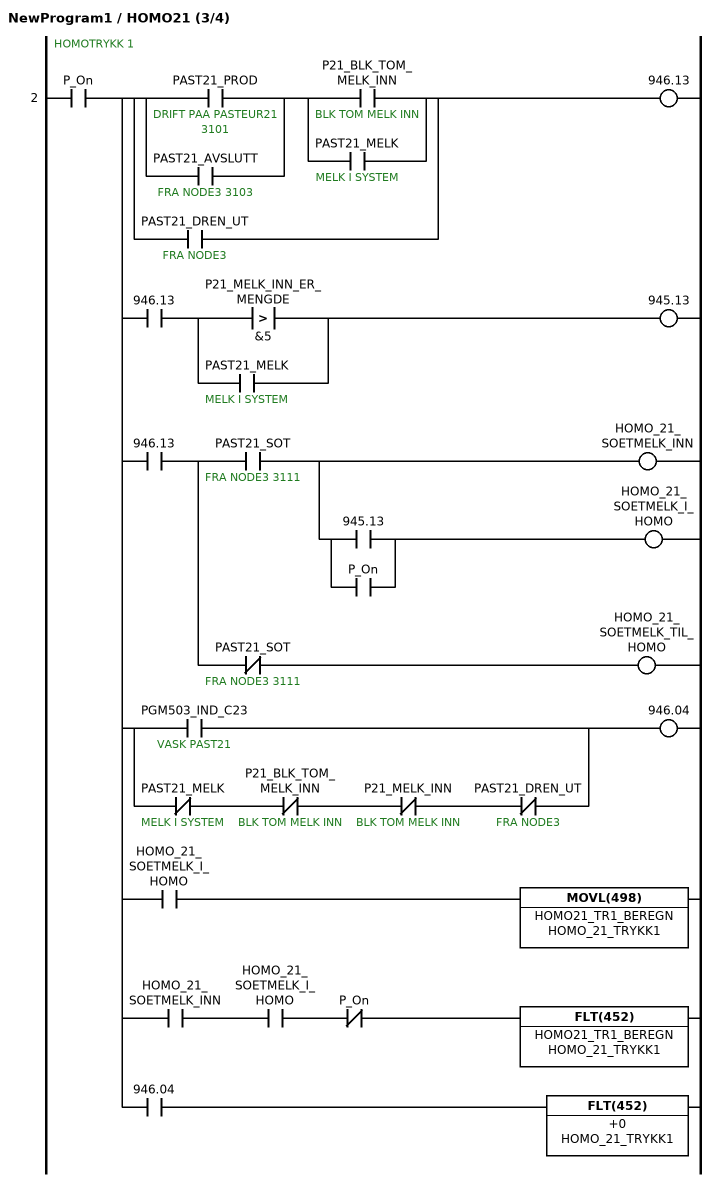
; [picture p1128: NewProgram1 / HOMO21, rungs 2-2]
; rung 2: HOMOTRYKK 1
LD P_On
OUT TR0
LD PAST21_PROD  ; DRIFT PAA PASTEUR21 3101
OR PAST21_AVSLUTT  ; FRA NODE3 3103
LD P21_BLK_TOM_MELK_INN  ; BLK TOM MELK INN
OR PAST21_MELK  ; MELK I SYSTEM
ANDLD
OR PAST21_DREN_UT  ; FRA NODE3
ANDLD
OUT 946.13
LD TR0
AND 946.13
LD>(320) P21_MELK_INN_ER_MENGDE &5
OR PAST21_MELK  ; MELK I SYSTEM
ANDLD
OUT 945.13
LD TR0
AND 946.13
OUT TR1
AND PAST21_SOT  ; FRA NODE3 3111
OUT HOMO_21_SOETMELK_INN
LD 945.13
OR P_On
ANDLD
OUT HOMO_21_SOETMELK_I_HOMO
LD TR1
ANDNOT PAST21_SOT  ; FRA NODE3 3111
OUT HOMO_21_SOETMELK_TIL_HOMO
LD TR0
LD PGM503_IND_C23  ; VASK PAST21
LDNOT PAST21_MELK  ; MELK I SYSTEM
ANDNOT P21_BLK_TOM_MELK_INN  ; BLK TOM MELK INN
ANDNOT P21_MELK_INN  ; BLK TOM MELK INN
ANDNOT PAST21_DREN_UT  ; FRA NODE3
ORLD
ANDLD
OUT 946.04
LD TR0
AND HOMO_21_SOETMELK_I_HOMO
MOVL(498) HOMO21_TR1_BEREGN HOMO_21_TRYKK1
LD TR0
AND HOMO_21_SOETMELK_INN
AND HOMO_21_SOETMELK_I_HOMO
ANDNOT P_On
FLT(452) HOMO21_TR1_BEREGN HOMO_21_TRYKK1
LD TR0
AND 946.04
FLT(452) +0 HOMO_21_TRYKK1

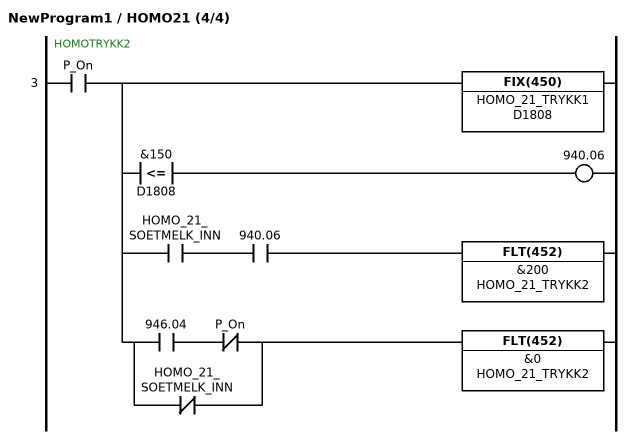
; rung 3: HOMOTRYKK2
LD P_On
OUT TR0
FIX(450) HOMO_21_TRYKK1 D1808
AND<=(315) &150 D1808
OUT 940.06
LD TR0
AND HOMO_21_SOETMELK_INN
AND 940.06
FLT(452) &200 HOMO_21_TRYKK2
LD TR0
LD 946.04
ANDNOT P_On
ORNOT HOMO_21_SOETMELK_INN
ANDLD
FLT(452) &0 HOMO_21_TRYKK2

### Section PAST22_TEMP_NIVÅ

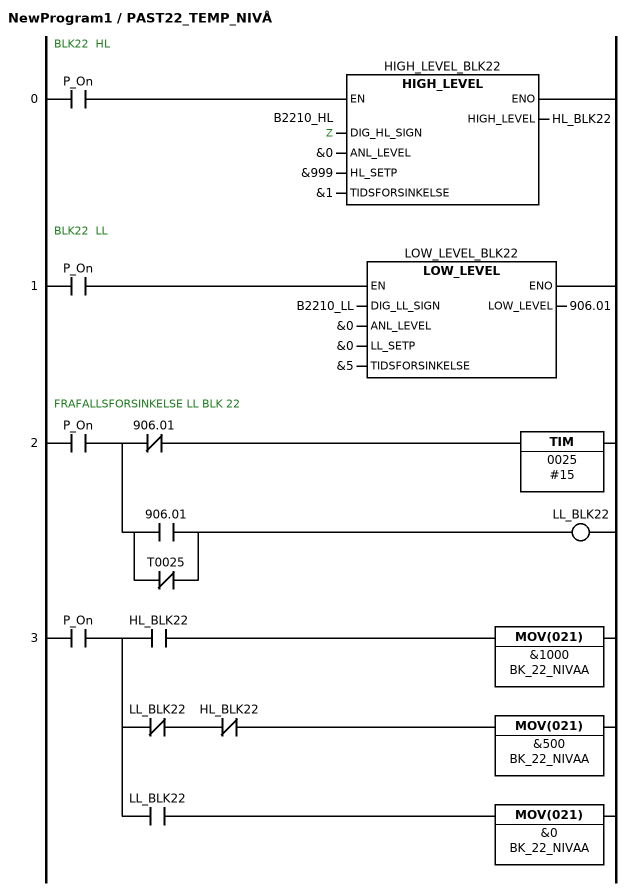
; rung 0: BLK22  HL
LD P_On
CALL HIGH_LEVEL_BLK22 : HIGH_LEVEL (DIG_HL_SIGN := B2210_HL, ANL_LEVEL := &0, HL_SETP := &999, TIDSFORSINKELSE := &1, HIGH_LEVEL => HL_BLK22)  ; Z
; rung 1: BLK22  LL
LD P_On
CALL LOW_LEVEL_BLK22 : LOW_LEVEL (DIG_LL_SIGN := B2210_LL, ANL_LEVEL := &0, LL_SETP := &0, TIDSFORSINKELSE := &5, LOW_LEVEL => 906.01)
; rung 2: FRAFALLSFORSINKELSE LL BLK 22
LD P_On
OUT TR0
ANDNOT 906.01
TIM 0025 #15
LD TR0
LD 906.01
ORNOT T0025
ANDLD
OUT LL_BLK22
; rung 3
LD P_On
OUT TR0
AND HL_BLK22
MOV(021) &1000 BK_22_NIVAA
LD TR0
ANDNOT LL_BLK22
ANDNOT HL_BLK22
MOV(021) &500 BK_22_NIVAA
LD TR0
AND LL_BLK22
MOV(021) &0 BK_22_NIVAA

### Section PAST22_DRIFT_OG_TYPE_MELK

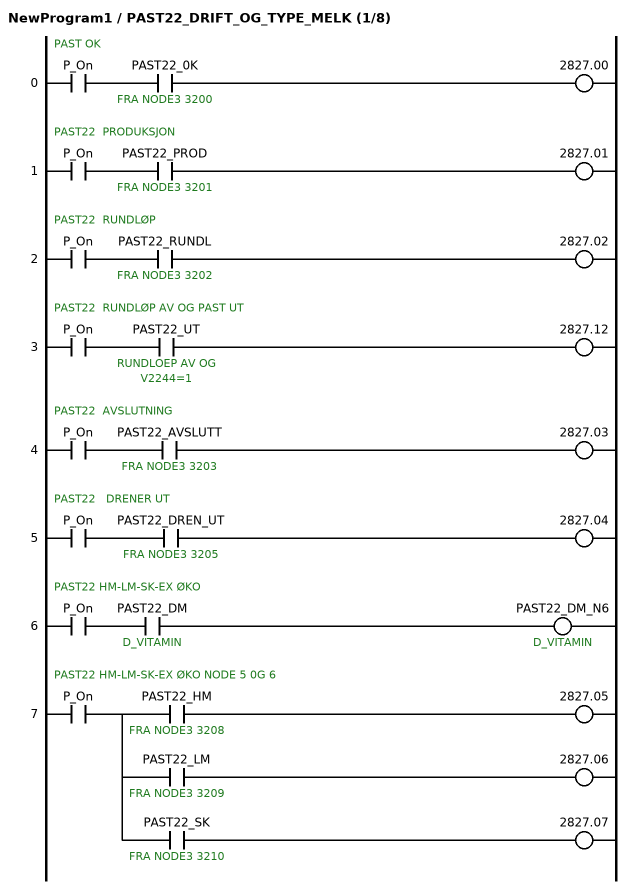
; rung 0: PAST OK
LD P_On
AND PAST22_0K  ; FRA NODE3 3200
OUT 2827.00
; rung 1: PAST22  PRODUKSJON
LD P_On
AND PAST22_PROD  ; FRA NODE3 3201
OUT 2827.01
; rung 2: PAST22  RUNDLØP
LD P_On
AND PAST22_RUNDL  ; FRA NODE3 3202
OUT 2827.02
; rung 3: PAST22  RUNDLØP AV OG PAST UT
LD P_On
AND PAST22_UT  ; RUNDLOEP AV OG V2244=1
OUT 2827.12
; rung 4: PAST22  AVSLUTNING
LD P_On
AND PAST22_AVSLUTT  ; FRA NODE3 3203
OUT 2827.03
; rung 5: PAST22   DRENER UT
LD P_On
AND PAST22_DREN_UT  ; FRA NODE3 3205
OUT 2827.04
; rung 6: PAST22 HM-LM-SK-EX ØKO
LD P_On
AND PAST22_DM  ; D_VITAMIN
OUT PAST22_DM_N6  ; D_VITAMIN
; rung 7: PAST22 HM-LM-SK-EX ØKO NODE 5 0G 6
LD P_On
OUT TR0
AND PAST22_HM  ; FRA NODE3 3208
OUT 2827.05
LD TR0
AND PAST22_LM  ; FRA NODE3 3209
OUT 2827.06
LD TR0
AND PAST22_SK  ; FRA NODE3 3210
OUT 2827.07

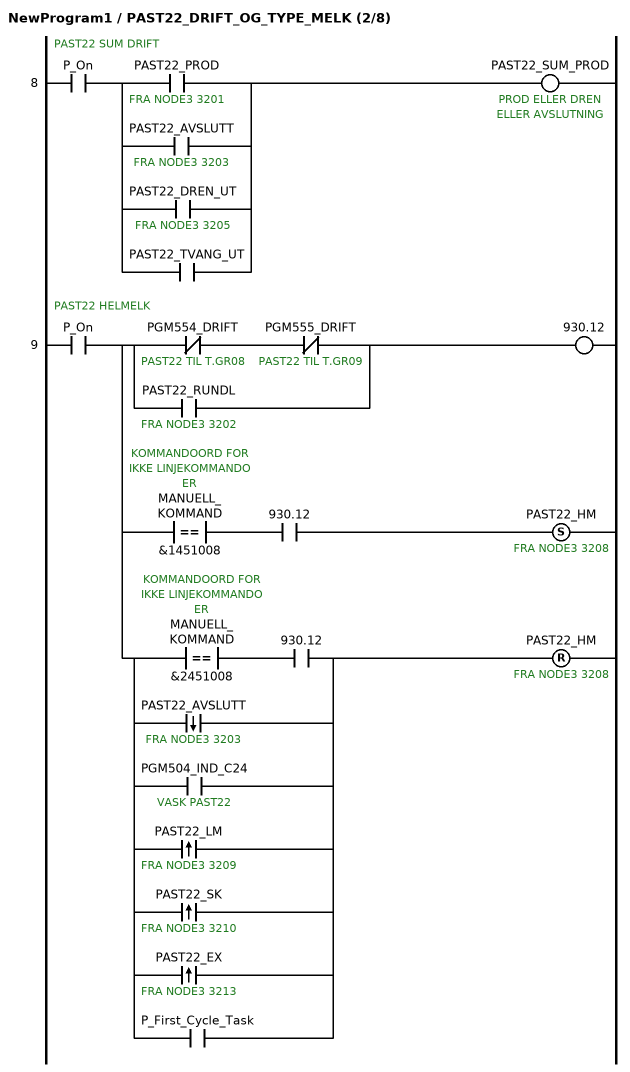
; rung 8: PAST22 SUM DRIFT
LD P_On
LD PAST22_PROD  ; FRA NODE3 3201
OR PAST22_AVSLUTT  ; FRA NODE3 3203
OR PAST22_DREN_UT  ; FRA NODE3 3205
OR PAST22_TVANG_UT
ANDLD
OUT PAST22_SUM_PROD  ; PROD ELLER DREN ELLER AVSLUTNING
; rung 9: PAST22 HELMELK
LD P_On
OUT TR0
LDNOT PGM554_DRIFT  ; PAST22 TIL T.GR08
ANDNOT PGM555_DRIFT  ; PAST22 TIL T.GR09
OR PAST22_RUNDL  ; FRA NODE3 3202
ANDLD
OUT 930.12
LD TR0
AND=L(301) MANUELL_KOMMAND &1451008  ; KOMMANDOORD FOR IKKE LINJEKOMMANDOER
AND 930.12
SET PAST22_HM  ; FRA NODE3 3208
LD TR0
LD=L(301) MANUELL_KOMMAND &2451008  ; KOMMANDOORD FOR IKKE LINJEKOMMANDOER
AND 930.12
%OR PAST22_AVSLUTT  ; FRA NODE3 3203
OR PGM504_IND_C24  ; VASK PAST22
@OR PAST22_LM  ; FRA NODE3 3209
@OR PAST22_SK  ; FRA NODE3 3210
@OR PAST22_EX  ; FRA NODE3 3213
OR P_First_Cycle_Task
ANDLD
RSET PAST22_HM  ; FRA NODE3 3208

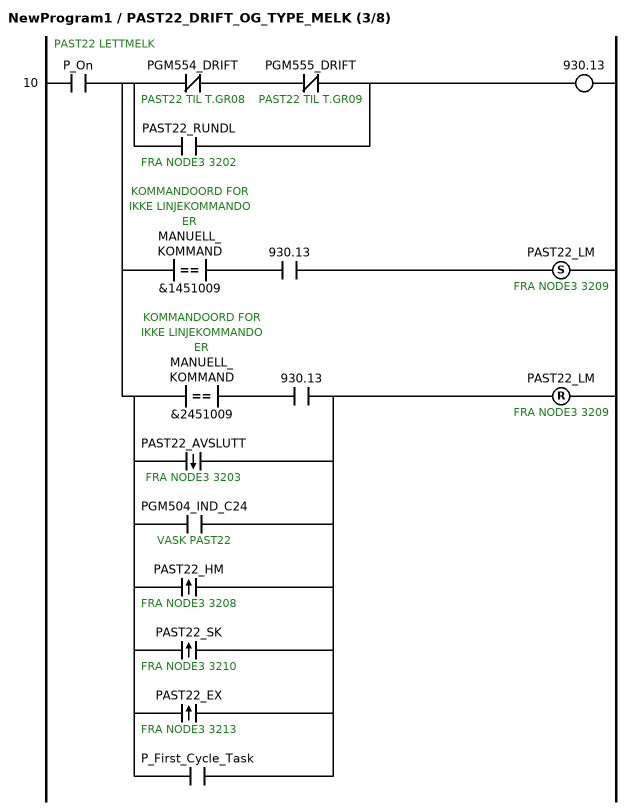
; rung 10: PAST22 LETTMELK
LD P_On
OUT TR0
LDNOT PGM554_DRIFT  ; PAST22 TIL T.GR08
ANDNOT PGM555_DRIFT  ; PAST22 TIL T.GR09
OR PAST22_RUNDL  ; FRA NODE3 3202
ANDLD
OUT 930.13
LD TR0
AND=L(301) MANUELL_KOMMAND &1451009  ; KOMMANDOORD FOR IKKE LINJEKOMMANDOER
AND 930.13
SET PAST22_LM  ; FRA NODE3 3209
LD TR0
LD=L(301) MANUELL_KOMMAND &2451009  ; KOMMANDOORD FOR IKKE LINJEKOMMANDOER
AND 930.13
%OR PAST22_AVSLUTT  ; FRA NODE3 3203
OR PGM504_IND_C24  ; VASK PAST22
@OR PAST22_HM  ; FRA NODE3 3208
@OR PAST22_SK  ; FRA NODE3 3210
@OR PAST22_EX  ; FRA NODE3 3213
OR P_First_Cycle_Task
ANDLD
RSET PAST22_LM  ; FRA NODE3 3209

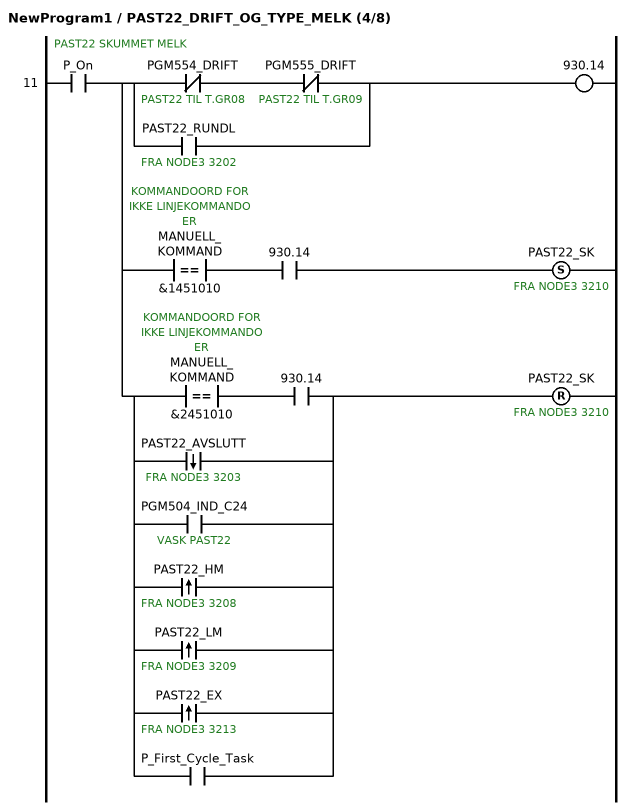
; rung 11: PAST22 SKUMMET MELK
LD P_On
OUT TR0
LDNOT PGM554_DRIFT  ; PAST22 TIL T.GR08
ANDNOT PGM555_DRIFT  ; PAST22 TIL T.GR09
OR PAST22_RUNDL  ; FRA NODE3 3202
ANDLD
OUT 930.14
LD TR0
AND=L(301) MANUELL_KOMMAND &1451010  ; KOMMANDOORD FOR IKKE LINJEKOMMANDOER
AND 930.14
SET PAST22_SK  ; FRA NODE3 3210
LD TR0
LD=L(301) MANUELL_KOMMAND &2451010  ; KOMMANDOORD FOR IKKE LINJEKOMMANDOER
AND 930.14
%OR PAST22_AVSLUTT  ; FRA NODE3 3203
OR PGM504_IND_C24  ; VASK PAST22
@OR PAST22_HM  ; FRA NODE3 3208
@OR PAST22_LM  ; FRA NODE3 3209
@OR PAST22_EX  ; FRA NODE3 3213
OR P_First_Cycle_Task
ANDLD
RSET PAST22_SK  ; FRA NODE3 3210

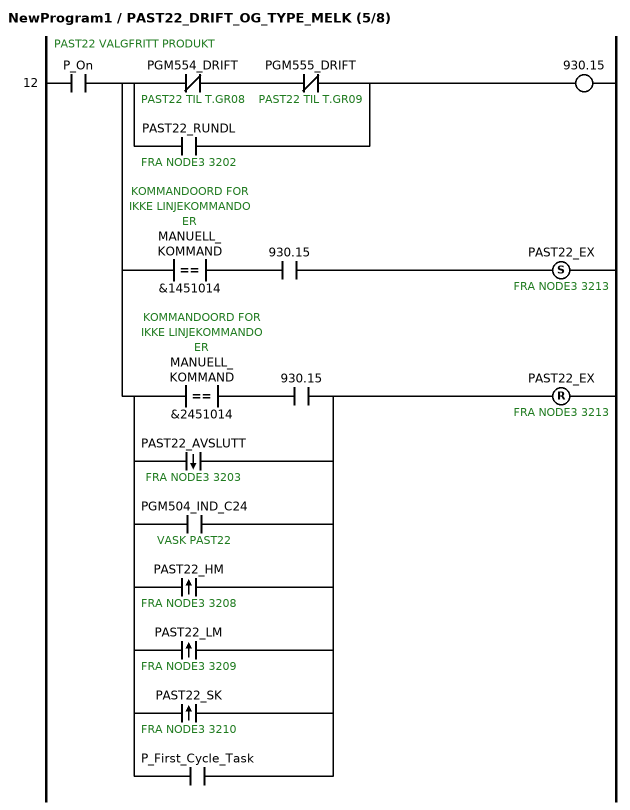
; rung 12: PAST22 VALGFRITT PRODUKT
LD P_On
OUT TR0
LDNOT PGM554_DRIFT  ; PAST22 TIL T.GR08
ANDNOT PGM555_DRIFT  ; PAST22 TIL T.GR09
OR PAST22_RUNDL  ; FRA NODE3 3202
ANDLD
OUT 930.15
LD TR0
AND=L(301) MANUELL_KOMMAND &1451014  ; KOMMANDOORD FOR IKKE LINJEKOMMANDOER
AND 930.15
SET PAST22_EX  ; FRA NODE3 3213
LD TR0
LD=L(301) MANUELL_KOMMAND &2451014  ; KOMMANDOORD FOR IKKE LINJEKOMMANDOER
AND 930.15
%OR PAST22_AVSLUTT  ; FRA NODE3 3203
OR PGM504_IND_C24  ; VASK PAST22
@OR PAST22_HM  ; FRA NODE3 3208
@OR PAST22_LM  ; FRA NODE3 3209
@OR PAST22_SK  ; FRA NODE3 3210
OR P_First_Cycle_Task
ANDLD
RSET PAST22_EX  ; FRA NODE3 3213

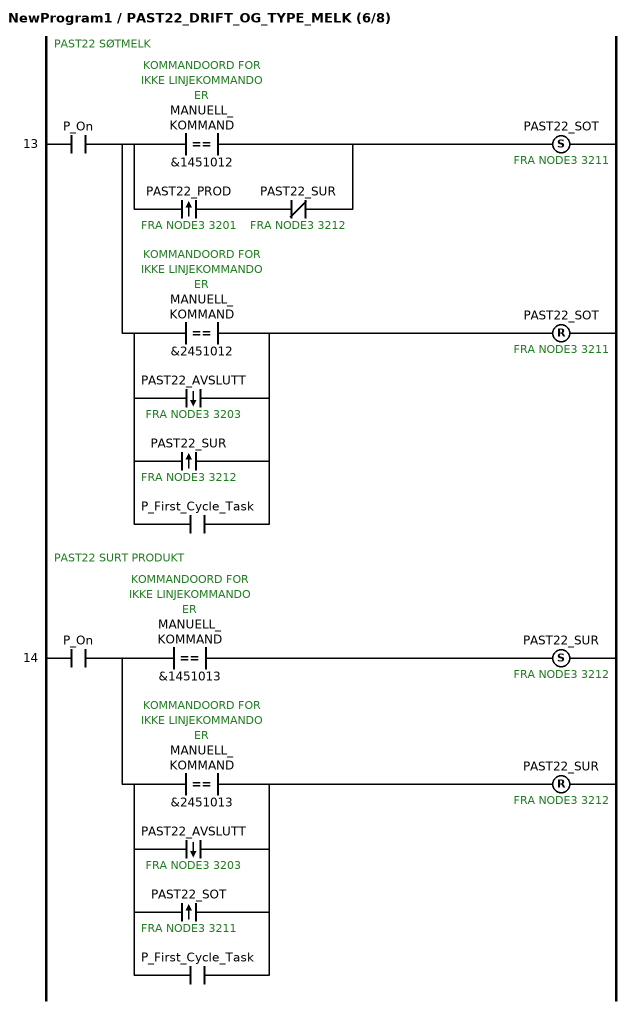
; rung 13: PAST22 SØTMELK
LD P_On
OUT TR0
LD=L(301) MANUELL_KOMMAND &1451012  ; KOMMANDOORD FOR IKKE LINJEKOMMANDOER
@LD PAST22_PROD  ; FRA NODE3 3201
ANDNOT PAST22_SUR  ; FRA NODE3 3212
ORLD
ANDLD
SET PAST22_SOT  ; FRA NODE3 3211
LD TR0
LD=L(301) MANUELL_KOMMAND &2451012  ; KOMMANDOORD FOR IKKE LINJEKOMMANDOER
%OR PAST22_AVSLUTT  ; FRA NODE3 3203
@OR PAST22_SUR  ; FRA NODE3 3212
OR P_First_Cycle_Task
ANDLD
RSET PAST22_SOT  ; FRA NODE3 3211
; rung 14: PAST22 SURT PRODUKT
LD P_On
OUT TR0
AND=L(301) MANUELL_KOMMAND &1451013  ; KOMMANDOORD FOR IKKE LINJEKOMMANDOER
SET PAST22_SUR  ; FRA NODE3 3212
LD TR0
LD=L(301) MANUELL_KOMMAND &2451013  ; KOMMANDOORD FOR IKKE LINJEKOMMANDOER
%OR PAST22_AVSLUTT  ; FRA NODE3 3203
@OR PAST22_SOT  ; FRA NODE3 3211
OR P_First_Cycle_Task
ANDLD
RSET PAST22_SUR  ; FRA NODE3 3212

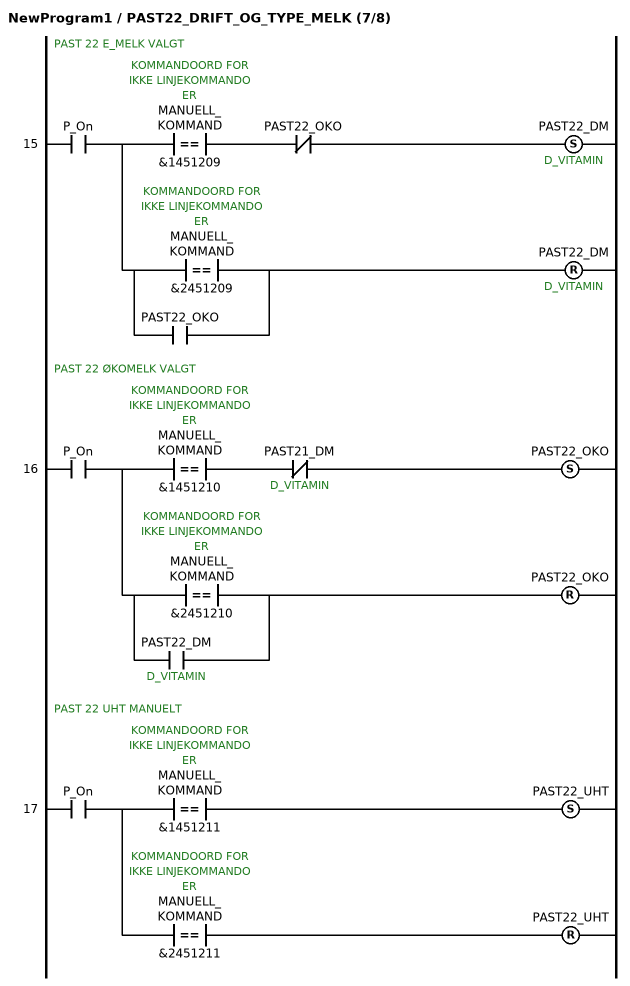
; rung 15: PAST 22 E_MELK VALGT
LD P_On
OUT TR0
AND=L(301) MANUELL_KOMMAND &1451209  ; KOMMANDOORD FOR IKKE LINJEKOMMANDOER
ANDNOT PAST22_OKO
SET PAST22_DM  ; D_VITAMIN
LD TR0
LD=L(301) MANUELL_KOMMAND &2451209  ; KOMMANDOORD FOR IKKE LINJEKOMMANDOER
OR PAST22_OKO
ANDLD
RSET PAST22_DM  ; D_VITAMIN
; rung 16: PAST 22 ØKOMELK VALGT
LD P_On
OUT TR0
AND=L(301) MANUELL_KOMMAND &1451210  ; KOMMANDOORD FOR IKKE LINJEKOMMANDOER
ANDNOT PAST21_DM  ; D_VITAMIN
SET PAST22_OKO
LD TR0
LD=L(301) MANUELL_KOMMAND &2451210  ; KOMMANDOORD FOR IKKE LINJEKOMMANDOER
OR PAST22_DM  ; D_VITAMIN
ANDLD
RSET PAST22_OKO
; rung 17: PAST 22 UHT MANUELT
LD P_On
OUT TR0
AND=L(301) MANUELL_KOMMAND &1451211  ; KOMMANDOORD FOR IKKE LINJEKOMMANDOER
SET PAST22_UHT
LD TR0
AND=L(301) MANUELL_KOMMAND &2451211  ; KOMMANDOORD FOR IKKE LINJEKOMMANDOER
RSET PAST22_UHT

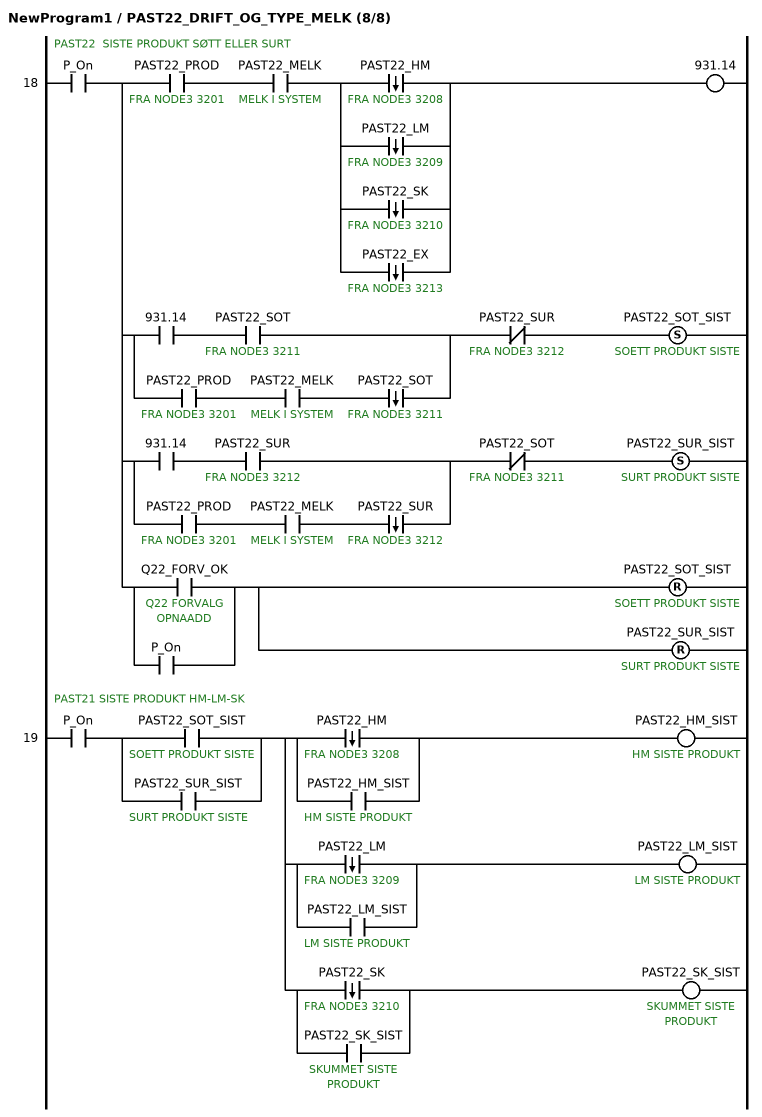
; rung 18: PAST22  SISTE PRODUKT SØTT ELLER SURT
LD P_On
OUT TR0
AND PAST22_PROD  ; FRA NODE3 3201
AND PAST22_MELK  ; MELK I SYSTEM
%LD PAST22_HM  ; FRA NODE3 3208
%OR PAST22_LM  ; FRA NODE3 3209
%OR PAST22_SK  ; FRA NODE3 3210
%OR PAST22_EX  ; FRA NODE3 3213
ANDLD
OUT 931.14
LD TR0
LD 931.14
AND PAST22_SOT  ; FRA NODE3 3211
LD PAST22_PROD  ; FRA NODE3 3201
AND PAST22_MELK  ; MELK I SYSTEM
%AND PAST22_SOT  ; FRA NODE3 3211
ORLD
ANDLD
ANDNOT PAST22_SUR  ; FRA NODE3 3212
SET PAST22_SOT_SIST  ; SOETT PRODUKT SISTE
LD TR0
LD 931.14
AND PAST22_SUR  ; FRA NODE3 3212
LD PAST22_PROD  ; FRA NODE3 3201
AND PAST22_MELK  ; MELK I SYSTEM
%AND PAST22_SUR  ; FRA NODE3 3212
ORLD
ANDLD
ANDNOT PAST22_SOT  ; FRA NODE3 3211
SET PAST22_SUR_SIST  ; SURT PRODUKT SISTE
LD TR0
LD Q22_FORV_OK  ; Q22 FORVALG OPNAADD
OR P_On
ANDLD
RSET PAST22_SOT_SIST  ; SOETT PRODUKT SISTE
RSET PAST22_SUR_SIST  ; SURT PRODUKT SISTE
; rung 19: PAST21 SISTE PRODUKT HM-LM-SK
LD P_On
LD PAST22_SOT_SIST  ; SOETT PRODUKT SISTE
OR PAST22_SUR_SIST  ; SURT PRODUKT SISTE
ANDLD
OUT TR0
%LD PAST22_HM  ; FRA NODE3 3208
OR PAST22_HM_SIST  ; HM SISTE PRODUKT
ANDLD
OUT PAST22_HM_SIST  ; HM SISTE PRODUKT
LD TR0
%LD PAST22_LM  ; FRA NODE3 3209
OR PAST22_LM_SIST  ; LM SISTE PRODUKT
ANDLD
OUT PAST22_LM_SIST  ; LM SISTE PRODUKT
LD TR0
%LD PAST22_SK  ; FRA NODE3 3210
OR PAST22_SK_SIST  ; SKUMMET SISTE PRODUKT
ANDLD
OUT PAST22_SK_SIST  ; SKUMMET SISTE PRODUKT

### Section PAST22_STATUSKONTROLL

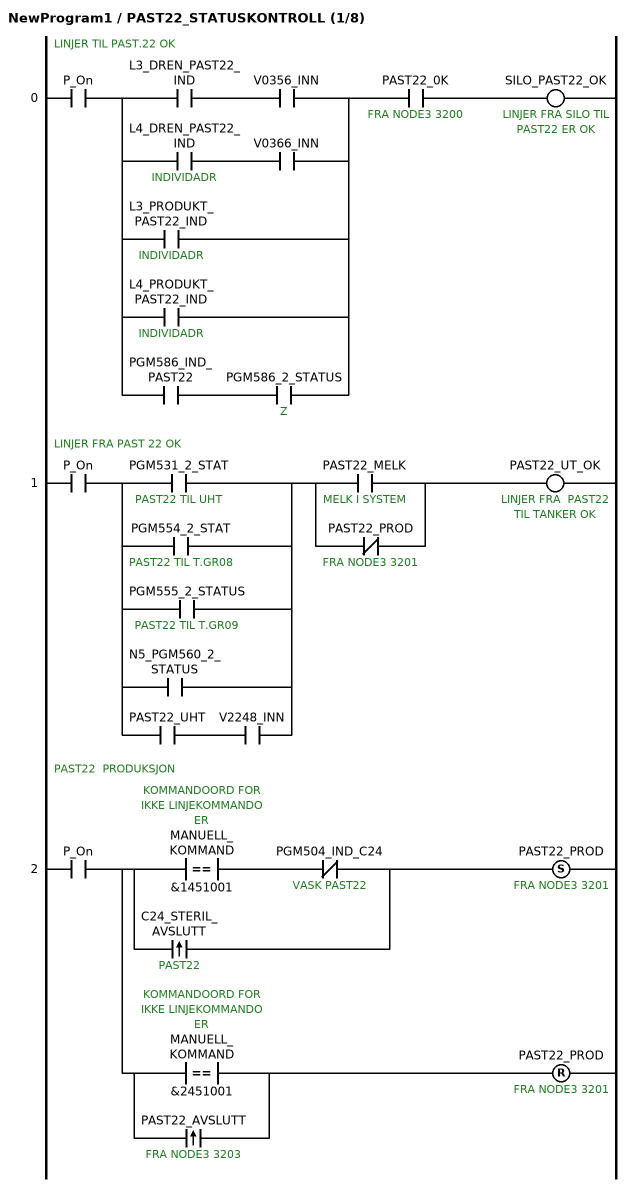
; rung 0: LINJER TIL PAST.22 OK
LD P_On
LD L3_DREN_PAST22_IND
AND V0356_INN
LD L4_DREN_PAST22_IND  ; INDIVIDADR
AND V0366_INN
ORLD
OR L3_PRODUKT_PAST22_IND  ; INDIVIDADR
OR L4_PRODUKT_PAST22_IND  ; INDIVIDADR
LD PGM586_IND_PAST22
AND PGM586_2_STATUS  ; Z
ORLD
ANDLD
AND PAST22_0K  ; FRA NODE3 3200
OUT SILO_PAST22_OK  ; LINJER FRA SILO TIL  PAST22 ER OK
; rung 1: LINJER FRA PAST 22 OK
LD P_On
LD PGM531_2_STAT  ; PAST22 TIL UHT
OR PGM554_2_STAT  ; PAST22 TIL T.GR08
OR PGM555_2_STATUS  ; PAST22 TIL T.GR09
OR N5_PGM560_2_STATUS
LD PAST22_UHT
AND V2248_INN
ORLD
ANDLD
LD PAST22_MELK  ; MELK I SYSTEM
ORNOT PAST22_PROD  ; FRA NODE3 3201
ANDLD
OUT PAST22_UT_OK  ; LINJER FRA  PAST22 TIL TANKER OK
; rung 2: PAST22  PRODUKSJON
LD P_On
OUT TR0
LD=L(301) MANUELL_KOMMAND &1451001  ; KOMMANDOORD FOR IKKE LINJEKOMMANDOER
ANDNOT PGM504_IND_C24  ; VASK PAST22
@OR C24_STERIL_AVSLUTT  ; PAST22
ANDLD
SET PAST22_PROD  ; FRA NODE3 3201
LD TR0
LD=L(301) MANUELL_KOMMAND &2451001  ; KOMMANDOORD FOR IKKE LINJEKOMMANDOER
@OR PAST22_AVSLUTT  ; FRA NODE3 3203
ANDLD
RSET PAST22_PROD  ; FRA NODE3 3201

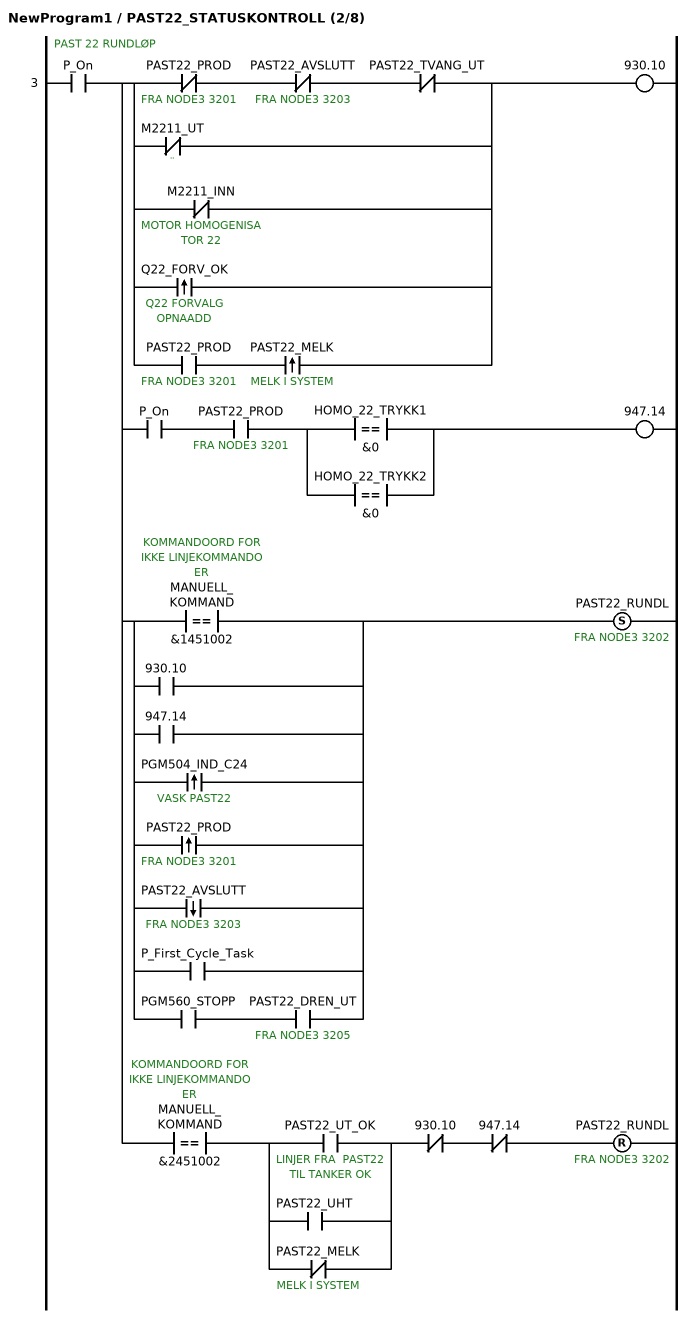
; rung 3: PAST 22 RUNDLØP
LD P_On
OUT TR0
LDNOT PAST22_PROD  ; FRA NODE3 3201
ANDNOT PAST22_AVSLUTT  ; FRA NODE3 3203
ANDNOT PAST22_TVANG_UT
ORNOT M2211_UT  ; ¨
ORNOT M2211_INN  ; MOTOR HOMOGENISATOR 22
@OR Q22_FORV_OK  ; Q22 FORVALG OPNAADD
LD PAST22_PROD  ; FRA NODE3 3201
@AND PAST22_MELK  ; MELK I SYSTEM
ORLD
ANDLD
OUT 930.10
LD TR0
AND P_On
AND PAST22_PROD  ; FRA NODE3 3201
LD=L(301) HOMO_22_TRYKK1 &0
OR=L(301) HOMO_22_TRYKK2 &0
ANDLD
OUT 947.14
LD TR0
LD=L(301) MANUELL_KOMMAND &1451002  ; KOMMANDOORD FOR IKKE LINJEKOMMANDOER
OR 930.10
OR 947.14
@OR PGM504_IND_C24  ; VASK PAST22
@OR PAST22_PROD  ; FRA NODE3 3201
%OR PAST22_AVSLUTT  ; FRA NODE3 3203
OR P_First_Cycle_Task
LD PGM560_STOPP
AND PAST22_DREN_UT  ; FRA NODE3 3205
ORLD
ANDLD
SET PAST22_RUNDL  ; FRA NODE3 3202
LD TR0
AND=L(301) MANUELL_KOMMAND &2451002  ; KOMMANDOORD FOR IKKE LINJEKOMMANDOER
LD PAST22_UT_OK  ; LINJER FRA  PAST22 TIL TANKER OK
OR PAST22_UHT
ORNOT PAST22_MELK  ; MELK I SYSTEM
ANDLD
ANDNOT 930.10
ANDNOT 947.14
RSET PAST22_RUNDL  ; FRA NODE3 3202

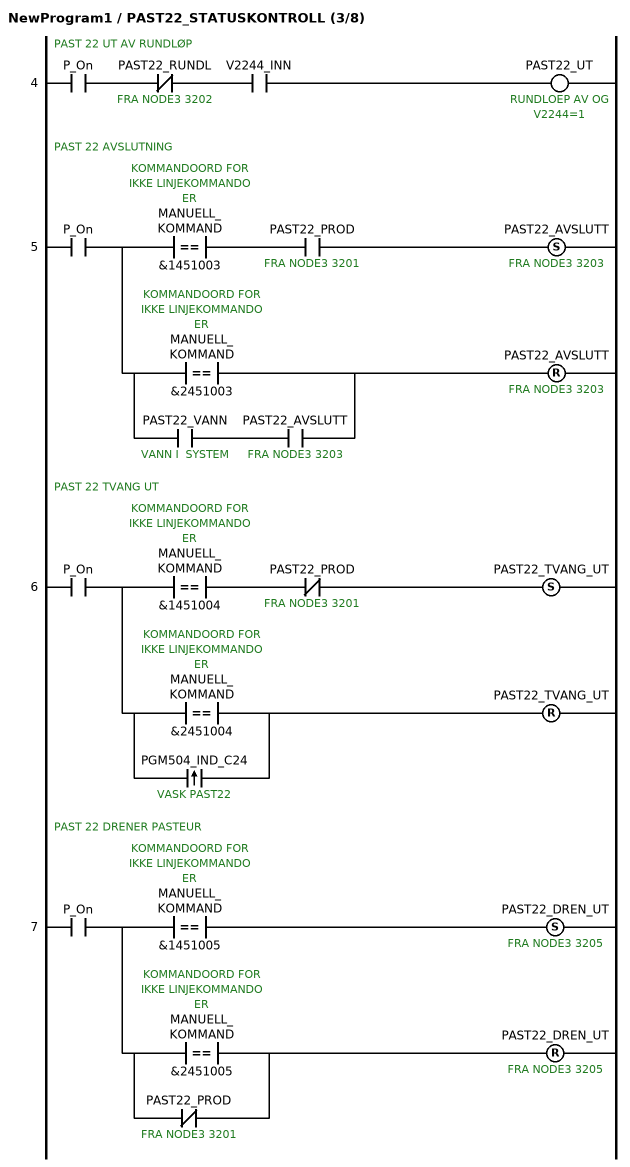
; rung 4: PAST 22 UT AV RUNDLØP
LD P_On
ANDNOT PAST22_RUNDL  ; FRA NODE3 3202
AND V2244_INN
OUT PAST22_UT  ; RUNDLOEP AV OG V2244=1
; rung 5: PAST 22 AVSLUTNING
LD P_On
OUT TR0
AND=L(301) MANUELL_KOMMAND &1451003  ; KOMMANDOORD FOR IKKE LINJEKOMMANDOER
AND PAST22_PROD  ; FRA NODE3 3201
SET PAST22_AVSLUTT  ; FRA NODE3 3203
LD TR0
LD=L(301) MANUELL_KOMMAND &2451003  ; KOMMANDOORD FOR IKKE LINJEKOMMANDOER
LD PAST22_VANN  ; VANN I  SYSTEM
AND PAST22_AVSLUTT  ; FRA NODE3 3203
ORLD
ANDLD
RSET PAST22_AVSLUTT  ; FRA NODE3 3203
; rung 6: PAST 22 TVANG UT
LD P_On
OUT TR0
AND=L(301) MANUELL_KOMMAND &1451004  ; KOMMANDOORD FOR IKKE LINJEKOMMANDOER
ANDNOT PAST22_PROD  ; FRA NODE3 3201
SET PAST22_TVANG_UT
LD TR0
LD=L(301) MANUELL_KOMMAND &2451004  ; KOMMANDOORD FOR IKKE LINJEKOMMANDOER
@OR PGM504_IND_C24  ; VASK PAST22
ANDLD
RSET PAST22_TVANG_UT
; rung 7: PAST 22 DRENER PASTEUR
LD P_On
OUT TR0
AND=L(301) MANUELL_KOMMAND &1451005  ; KOMMANDOORD FOR IKKE LINJEKOMMANDOER
SET PAST22_DREN_UT  ; FRA NODE3 3205
LD TR0
LD=L(301) MANUELL_KOMMAND &2451005  ; KOMMANDOORD FOR IKKE LINJEKOMMANDOER
ORNOT PAST22_PROD  ; FRA NODE3 3201
ANDLD
RSET PAST22_DREN_UT  ; FRA NODE3 3205

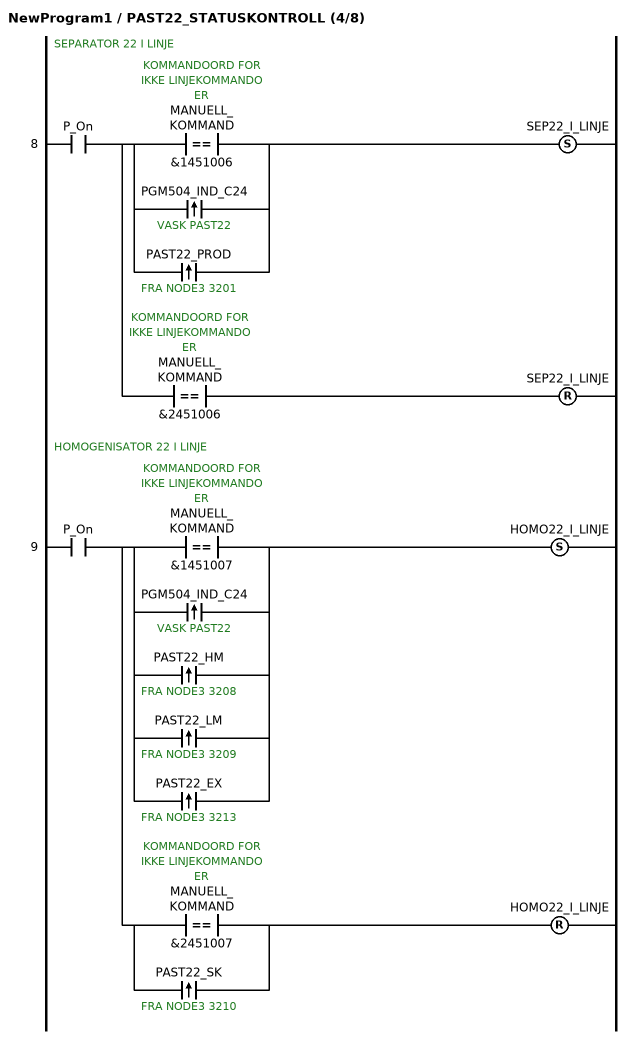
; rung 8: SEPARATOR 22 I LINJE
LD P_On
OUT TR0
LD=L(301) MANUELL_KOMMAND &1451006  ; KOMMANDOORD FOR IKKE LINJEKOMMANDOER
@OR PGM504_IND_C24  ; VASK PAST22
@OR PAST22_PROD  ; FRA NODE3 3201
ANDLD
SET SEP22_I_LINJE
LD TR0
AND=L(301) MANUELL_KOMMAND &2451006  ; KOMMANDOORD FOR IKKE LINJEKOMMANDOER
RSET SEP22_I_LINJE
; rung 9: HOMOGENISATOR 22 I LINJE
LD P_On
OUT TR0
LD=L(301) MANUELL_KOMMAND &1451007  ; KOMMANDOORD FOR IKKE LINJEKOMMANDOER
@OR PGM504_IND_C24  ; VASK PAST22
@OR PAST22_HM  ; FRA NODE3 3208
@OR PAST22_LM  ; FRA NODE3 3209
@OR PAST22_EX  ; FRA NODE3 3213
ANDLD
SET HOMO22_I_LINJE
LD TR0
LD=L(301) MANUELL_KOMMAND &2451007  ; KOMMANDOORD FOR IKKE LINJEKOMMANDOER
@OR PAST22_SK  ; FRA NODE3 3210
ANDLD
RSET HOMO22_I_LINJE

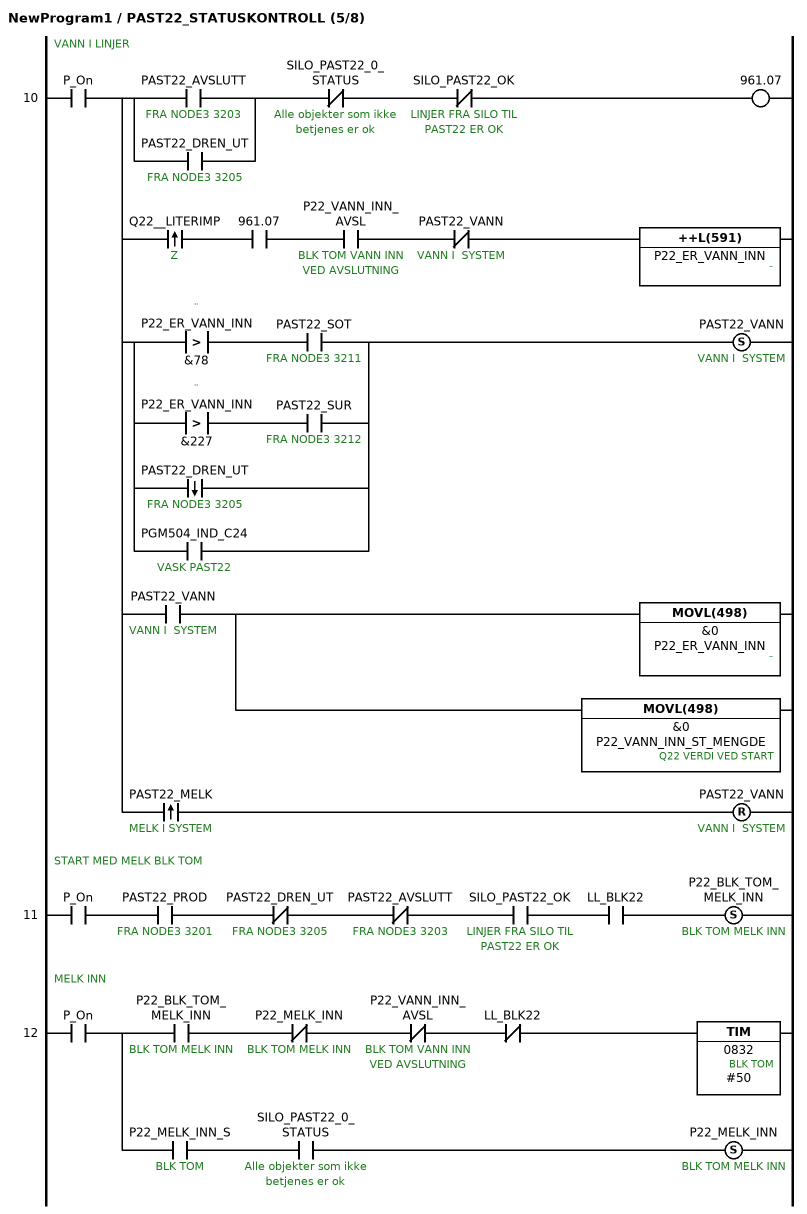
; rung 10: VANN I LINJER
LD P_On
OUT TR0
LD PAST22_AVSLUTT  ; FRA NODE3 3203
OR PAST22_DREN_UT  ; FRA NODE3 3205
ANDLD
ANDNOT SILO_PAST22_0_STATUS  ; Alle objekter som ikke betjenes er ok
ANDNOT SILO_PAST22_OK  ; LINJER FRA SILO TIL  PAST22 ER OK
OUT 961.07
LD TR0
@AND Q22__LITERIMP  ; Z
AND 961.07
AND P22_VANN_INN_AVSL  ; BLK TOM VANN INN VED AVSLUTNING
ANDNOT PAST22_VANN  ; VANN I  SYSTEM
++L(591) P22_ER_VANN_INN  ; ¨
LD TR0
LD>L(321) P22_ER_VANN_INN &78  ; ¨
AND PAST22_SOT  ; FRA NODE3 3211
LD>L(321) P22_ER_VANN_INN &227  ; ¨
AND PAST22_SUR  ; FRA NODE3 3212
ORLD
%OR PAST22_DREN_UT  ; FRA NODE3 3205
OR PGM504_IND_C24  ; VASK PAST22
ANDLD
SET PAST22_VANN  ; VANN I  SYSTEM
LD TR0
AND PAST22_VANN  ; VANN I  SYSTEM
MOVL(498) &0 P22_ER_VANN_INN  ; ¨
MOVL(498) &0 P22_VANN_INN_ST_MENGDE  ; Q22 VERDI VED START
LD TR0
@AND PAST22_MELK  ; MELK I SYSTEM
RSET PAST22_VANN  ; VANN I  SYSTEM
; rung 11: START MED MELK BLK TOM
LD P_On
AND PAST22_PROD  ; FRA NODE3 3201
ANDNOT PAST22_DREN_UT  ; FRA NODE3 3205
ANDNOT PAST22_AVSLUTT  ; FRA NODE3 3203
AND SILO_PAST22_OK  ; LINJER FRA SILO TIL  PAST22 ER OK
AND LL_BLK22
SET P22_BLK_TOM_MELK_INN  ; BLK TOM MELK INN
; rung 12: MELK INN
LD P_On
OUT TR0
AND P22_BLK_TOM_MELK_INN  ; BLK TOM MELK INN
ANDNOT P22_MELK_INN  ; BLK TOM MELK INN
ANDNOT P22_VANN_INN_AVSL  ; BLK TOM VANN INN VED AVSLUTNING
ANDNOT LL_BLK22
TIM 0832 #50  ; BLK TOM
LD TR0
AND P22_MELK_INN_S  ; BLK TOM
AND SILO_PAST22_0_STATUS  ; Alle objekter som ikke betjenes er ok
SET P22_MELK_INN  ; BLK TOM MELK INN

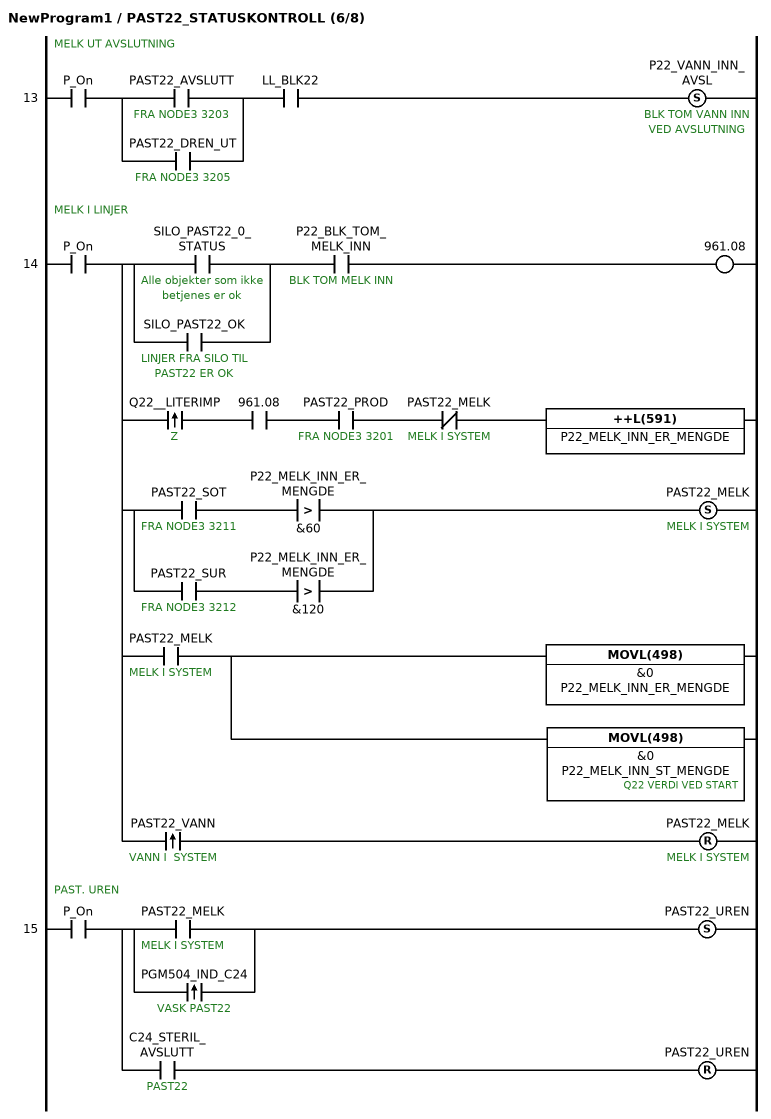
; rung 13: MELK UT AVSLUTNING
LD P_On
LD PAST22_AVSLUTT  ; FRA NODE3 3203
OR PAST22_DREN_UT  ; FRA NODE3 3205
ANDLD
AND LL_BLK22
SET P22_VANN_INN_AVSL  ; BLK TOM VANN INN VED AVSLUTNING
; rung 14: MELK I LINJER
LD P_On
OUT TR0
LD SILO_PAST22_0_STATUS  ; Alle objekter som ikke betjenes er ok
OR SILO_PAST22_OK  ; LINJER FRA SILO TIL  PAST22 ER OK
ANDLD
AND P22_BLK_TOM_MELK_INN  ; BLK TOM MELK INN
OUT 961.08
LD TR0
@AND Q22__LITERIMP  ; Z
AND 961.08
AND PAST22_PROD  ; FRA NODE3 3201
ANDNOT PAST22_MELK  ; MELK I SYSTEM
++L(591) P22_MELK_INN_ER_MENGDE
LD TR0
LD PAST22_SOT  ; FRA NODE3 3211
AND>L(321) P22_MELK_INN_ER_MENGDE &60
LD PAST22_SUR  ; FRA NODE3 3212
AND>L(321) P22_MELK_INN_ER_MENGDE &120
ORLD
ANDLD
SET PAST22_MELK  ; MELK I SYSTEM
LD TR0
AND PAST22_MELK  ; MELK I SYSTEM
MOVL(498) &0 P22_MELK_INN_ER_MENGDE
MOVL(498) &0 P22_MELK_INN_ST_MENGDE  ; Q22 VERDI VED START
LD TR0
@AND PAST22_VANN  ; VANN I  SYSTEM
RSET PAST22_MELK  ; MELK I SYSTEM
; rung 15: PAST. UREN
LD P_On
OUT TR0
LD PAST22_MELK  ; MELK I SYSTEM
@OR PGM504_IND_C24  ; VASK PAST22
ANDLD
SET PAST22_UREN
LD TR0
AND C24_STERIL_AVSLUTT  ; PAST22
RSET PAST22_UREN

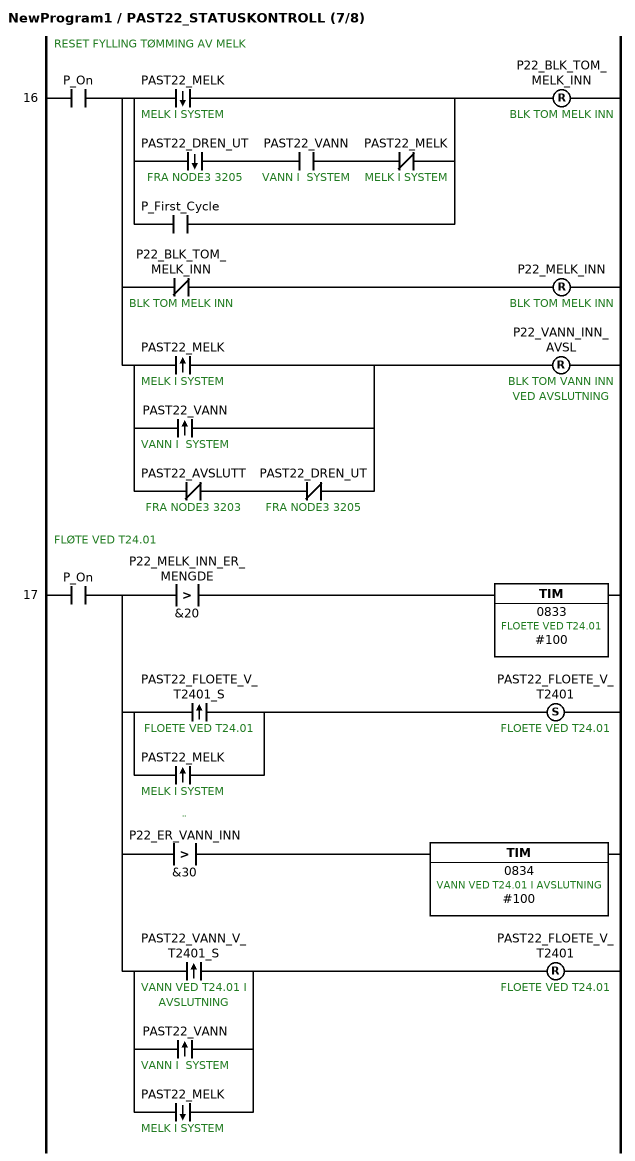
; rung 16: RESET FYLLING TØMMING AV MELK
LD P_On
OUT TR0
%LD PAST22_MELK  ; MELK I SYSTEM
%LD PAST22_DREN_UT  ; FRA NODE3 3205
AND PAST22_VANN  ; VANN I  SYSTEM
ANDNOT PAST22_MELK  ; MELK I SYSTEM
ORLD
OR P_First_Cycle
ANDLD
RSET P22_BLK_TOM_MELK_INN  ; BLK TOM MELK INN
LD TR0
ANDNOT P22_BLK_TOM_MELK_INN  ; BLK TOM MELK INN
RSET P22_MELK_INN  ; BLK TOM MELK INN
LD TR0
@LD PAST22_MELK  ; MELK I SYSTEM
@OR PAST22_VANN  ; VANN I  SYSTEM
LDNOT PAST22_AVSLUTT  ; FRA NODE3 3203
ANDNOT PAST22_DREN_UT  ; FRA NODE3 3205
ORLD
ANDLD
RSET P22_VANN_INN_AVSL  ; BLK TOM VANN INN VED AVSLUTNING
; rung 17: FLØTE VED T24.01
LD P_On
OUT TR0
AND>L(321) P22_MELK_INN_ER_MENGDE &20
TIM 0833 #100  ; FLOETE VED T24.01
LD TR0
@LD PAST22_FLOETE_V_T2401_S  ; FLOETE VED T24.01
@OR PAST22_MELK  ; MELK I SYSTEM
ANDLD
SET PAST22_FLOETE_V_T2401  ; FLOETE VED T24.01
LD TR0
AND>L(321) P22_ER_VANN_INN &30  ; ¨
TIM 0834 #100  ; VANN VED T24.01 I AVSLUTNING
LD TR0
@LD PAST22_VANN_V_T2401_S  ; VANN VED T24.01 I AVSLUTNING
@OR PAST22_VANN  ; VANN I  SYSTEM
%OR PAST22_MELK  ; MELK I SYSTEM
ANDLD
RSET PAST22_FLOETE_V_T2401  ; FLOETE VED T24.01

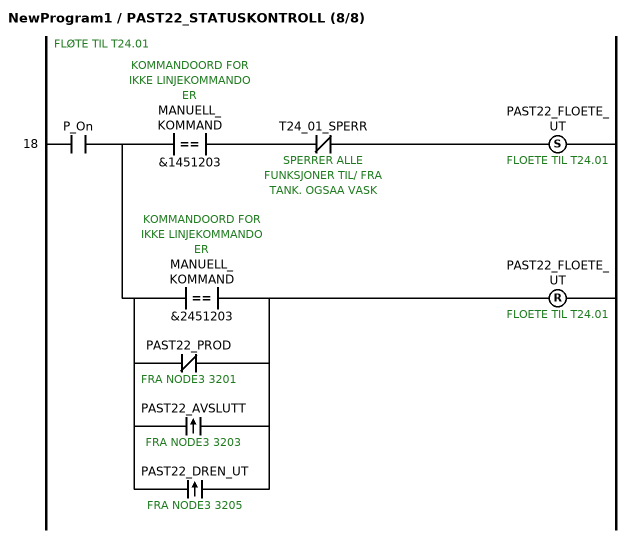
; rung 18: FLØTE TIL T24.01
LD P_On
OUT TR0
AND=L(301) MANUELL_KOMMAND &1451203  ; KOMMANDOORD FOR IKKE LINJEKOMMANDOER
ANDNOT T24_01_SPERR  ; SPERRER ALLE FUNKSJONER TIL/ FRA TANK. OGSAA VASK
SET PAST22_FLOETE_UT  ; FLOETE TIL T24.01
LD TR0
LD=L(301) MANUELL_KOMMAND &2451203  ; KOMMANDOORD FOR IKKE LINJEKOMMANDOER
ORNOT PAST22_PROD  ; FRA NODE3 3201
@OR PAST22_AVSLUTT  ; FRA NODE3 3203
@OR PAST22_DREN_UT  ; FRA NODE3 3205
ANDLD
RSET PAST22_FLOETE_UT  ; FLOETE TIL T24.01

### Section PAST22_OMSLAGSKONTROLL

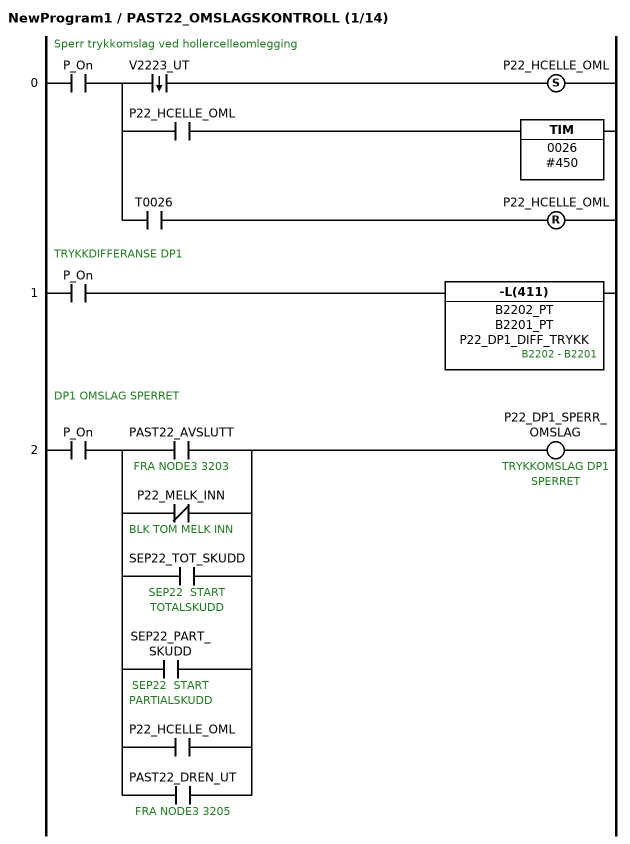
; rung 0: Sperr trykkomslag ved hollercelleomlegging
LD P_On
OUT TR0
%AND V2223_UT
SET P22_HCELLE_OML
LD TR0
AND P22_HCELLE_OML
TIM 0026 #450
LD TR0
AND T0026
RSET P22_HCELLE_OML
; rung 1: TRYKKDIFFERANSE DP1
LD P_On
-L(411) B2202_PT B2201_PT P22_DP1_DIFF_TRYKK  ; B2202 - B2201
; rung 2: DP1 OMSLAG SPERRET
LD P_On  // CF113 INVERTERES OM SPERRING AV OMSLAG VED DP1 SKAL OPPHEVES
LD PAST22_AVSLUTT  ; FRA NODE3 3203
ORNOT P22_MELK_INN  ; BLK TOM MELK INN
OR SEP22_TOT_SKUDD  ; SEP22  START TOTALSKUDD
OR SEP22_PART_SKUDD  ; SEP22  START PARTIALSKUDD
OR P22_HCELLE_OML
OR PAST22_DREN_UT  ; FRA NODE3 3205
ANDLD
OUT P22_DP1_SPERR_OMSLAG  ; TRYKKOMSLAG DP1 SPERRET

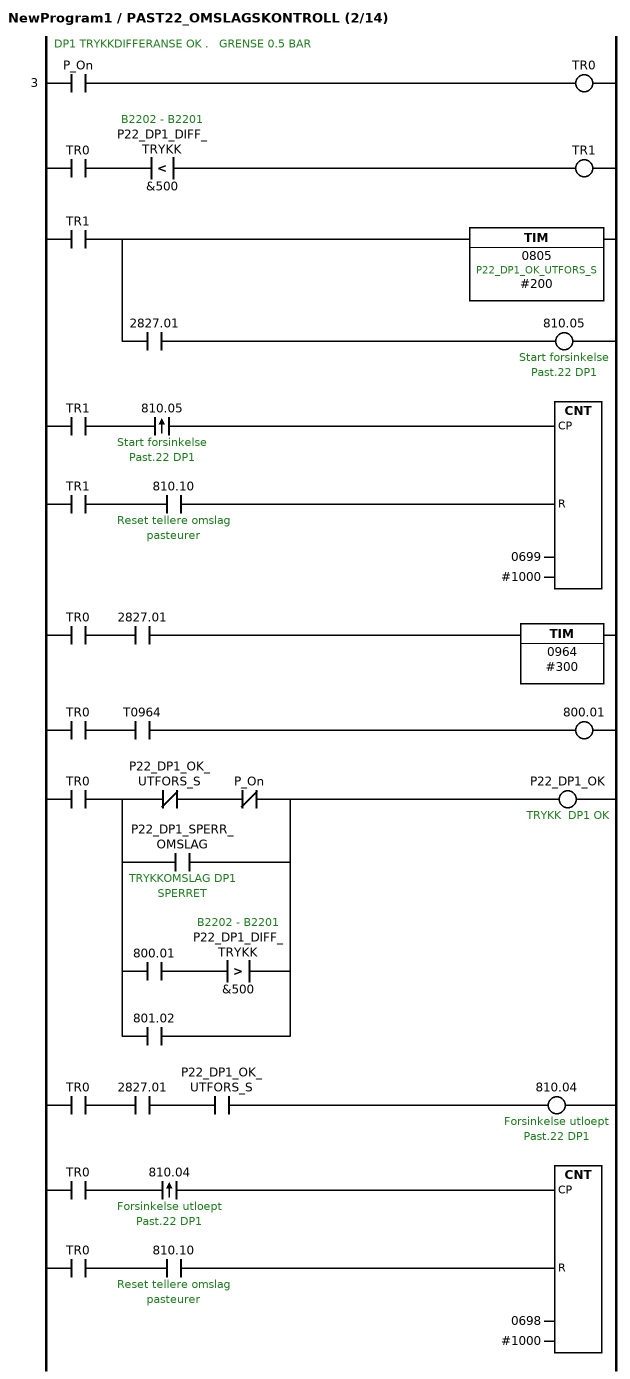
; rung 3: DP1 TRYKKDIFFERANSE OK .   GRENSE 0.5 BAR
LD P_On
OUT TR0
AND<SL(313) P22_DP1_DIFF_TRYKK &500  ; B2202 - B2201
OUT TR1
TIM 0805 #200  ; P22_DP1_OK_UTFORS_S
AND 2827.01
OUT 810.05  ; Start forsinkelse Past.22 DP1
LD TR1
@AND 810.05  ; Start forsinkelse Past.22 DP1
LD TR1
AND 810.10  ; Reset tellere omslag pasteurer
CNT 0699 #1000
LD TR0
AND 2827.01
TIM 0964 #300
LD TR0
AND T0964
OUT 800.01
LD TR0
LDNOT P22_DP1_OK_UTFORS_S
ANDNOT P_On
OR P22_DP1_SPERR_OMSLAG  ; TRYKKOMSLAG DP1 SPERRET
LD 800.01
AND>SL(323) P22_DP1_DIFF_TRYKK &500  ; B2202 - B2201
ORLD
OR 801.02
ANDLD
OUT P22_DP1_OK  ; TRYKK  DP1 OK
LD TR0
AND 2827.01
AND P22_DP1_OK_UTFORS_S
OUT 810.04  ; Forsinkelse utloept Past.22 DP1
LD TR0
@AND 810.04  ; Forsinkelse utloept Past.22 DP1
LD TR0
AND 810.10  ; Reset tellere omslag pasteurer
CNT 0698 #1000

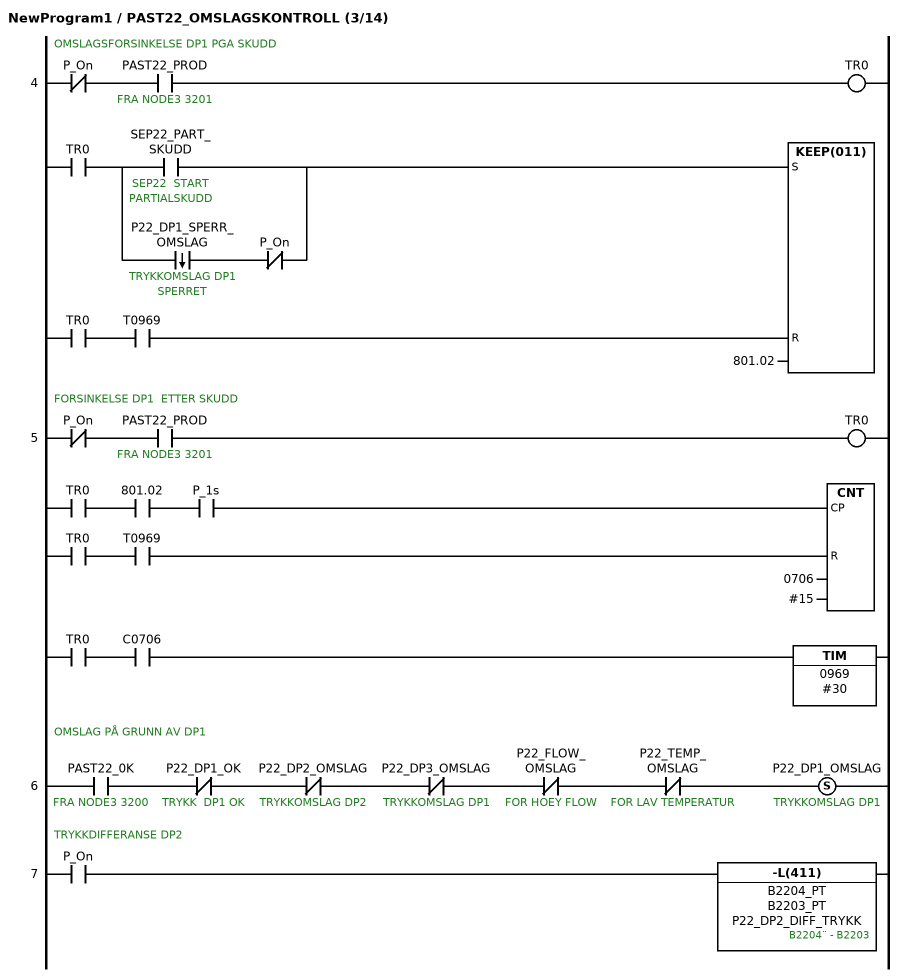
; rung 4: OMSLAGSFORSINKELSE DP1 PGA SKUDD
LDNOT P_On
AND PAST22_PROD  ; FRA NODE3 3201
OUT TR0
LD SEP22_PART_SKUDD  ; SEP22  START PARTIALSKUDD
%LD P22_DP1_SPERR_OMSLAG  ; TRYKKOMSLAG DP1 SPERRET
ANDNOT P_On
ORLD
ANDLD
LD TR0
AND T0969
KEEP(011) 801.02
; rung 5: FORSINKELSE DP1  ETTER SKUDD
LDNOT P_On
AND PAST22_PROD  ; FRA NODE3 3201
OUT TR0
AND 801.02
AND P_1s
LD TR0
AND T0969
CNT 0706 #15
LD TR0
AND C0706
TIM 0969 #30
; rung 6: OMSLAG PÅ GRUNN AV DP1
LD PAST22_0K  ; FRA NODE3 3200
ANDNOT P22_DP1_OK  ; TRYKK  DP1 OK
ANDNOT P22_DP2_OMSLAG  ; TRYKKOMSLAG DP2
ANDNOT P22_DP3_OMSLAG  ; TRYKKOMSLAG DP1
ANDNOT P22_FLOW_OMSLAG  ; FOR HOEY FLOW
ANDNOT P22_TEMP_OMSLAG  ; FOR LAV TEMPERATUR
SET P22_DP1_OMSLAG  ; TRYKKOMSLAG DP1
; rung 7: TRYKKDIFFERANSE DP2
LD P_On
-L(411) B2204_PT B2203_PT P22_DP2_DIFF_TRYKK  ; B2204¨ - B2203

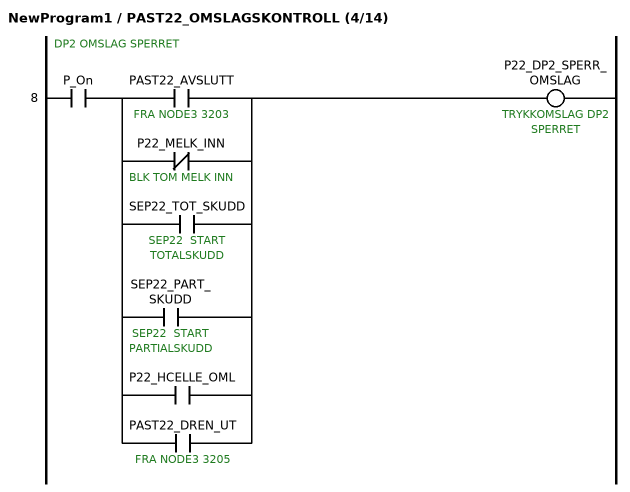
; rung 8: DP2 OMSLAG SPERRET
LD P_On  // CF113 INVERTERES OM SPERRING AV OMSLAG VED DP2 SKAL OPPHEVES
LD PAST22_AVSLUTT  ; FRA NODE3 3203
ORNOT P22_MELK_INN  ; BLK TOM MELK INN
OR SEP22_TOT_SKUDD  ; SEP22  START TOTALSKUDD
OR SEP22_PART_SKUDD  ; SEP22  START PARTIALSKUDD
OR P22_HCELLE_OML
OR PAST22_DREN_UT  ; FRA NODE3 3205
ANDLD
OUT P22_DP2_SPERR_OMSLAG  ; TRYKKOMSLAG DP2  SPERRET

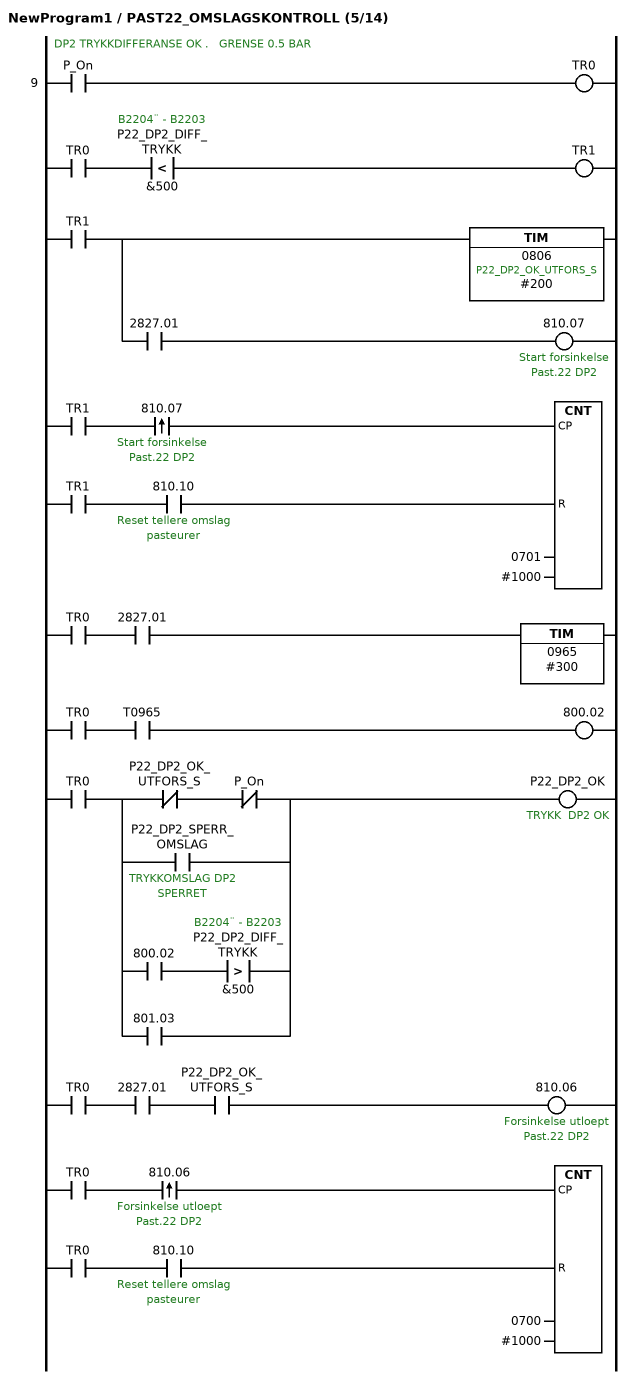
; rung 9: DP2 TRYKKDIFFERANSE OK .   GRENSE 0.5 BAR
LD P_On
OUT TR0
AND<SL(313) P22_DP2_DIFF_TRYKK &500  ; B2204¨ - B2203
OUT TR1
TIM 0806 #200  ; P22_DP2_OK_UTFORS_S
AND 2827.01
OUT 810.07  ; Start forsinkelse Past.22 DP2
LD TR1
@AND 810.07  ; Start forsinkelse Past.22 DP2
LD TR1
AND 810.10  ; Reset tellere omslag pasteurer
CNT 0701 #1000
LD TR0
AND 2827.01
TIM 0965 #300
LD TR0
AND T0965
OUT 800.02
LD TR0
LDNOT P22_DP2_OK_UTFORS_S
ANDNOT P_On
OR P22_DP2_SPERR_OMSLAG  ; TRYKKOMSLAG DP2  SPERRET
LD 800.02
AND>SL(323) P22_DP2_DIFF_TRYKK &500  ; B2204¨ - B2203
ORLD
OR 801.03
ANDLD
OUT P22_DP2_OK  ; TRYKK  DP2 OK
LD TR0
AND 2827.01
AND P22_DP2_OK_UTFORS_S
OUT 810.06  ; Forsinkelse utloept Past.22 DP2
LD TR0
@AND 810.06  ; Forsinkelse utloept Past.22 DP2
LD TR0
AND 810.10  ; Reset tellere omslag pasteurer
CNT 0700 #1000

